TYPE ST_timer :
STRUCT
END_STRUCT
END_TYPE

(* stored: Version 1.1.0.1, ProductVersion 3.1.4024.12
   DUT ST_timer: Id {e23d42df-24a4-4959-9633-c893292811c6} *)
